(*			
	EVERDE sp. z o.o.
	Rafał Osajda		08.08.2025		TC 4024.66
	Interfejs do wyciągania z SPM przez HMI danych do wyświetlania - dla ramki alarmy
*)
INTERFACE ITF_SPM_HMI_03_Lacznik EXTENDS  B_Baza.ITF_ZrodloIdentyfikacji

METHOD PrzygotujDaneDoWyswietleniaZgloszen : BOOL
VAR_INPUT

END_VAR
END_METHOD

METHOD PUBLIC ZwrocCzySaNoweZgloszeniaWSystemie : BOOL
VAR_INPUT
END_VAR
END_METHOD

END_INTERFACE

(* stored: Version 1.1.0.1
   Itf ITF_SPM_HMI_03_Lacznik: Id {c0fcb566-d7a2-0f1f-2e42-6e3bcadadae8}
   Method PrzygotujDaneDoWyswietleniaZgloszen: Id {0c125976-5e77-05e4-2fc9-a464ca4dd93f}
   Method ZwrocCzySaNoweZgloszeniaWSystemie: Id {7aaf3199-451a-017f-168b-7ff14b5d95ae} *)
